// TIA Portal V16 export
// export: Created 2022-01-12T14:34:29.5419654Z, ExportSetting WithDefaults, DisplayName Totally Integrated Automation Portal, DisplayVersion V16 Update 4, DisplayName TIA Portal Version Control Interface, DisplayVersion V16 Update 2, DisplayName TIA Portal Openness, DisplayVersion V16 Update 4, DisplayName STEP 7 Professional, DisplayVersion V16 Update 4, DisplayName STEP 7 Safety, DisplayVersion V16, DisplayName WinCC Professional, DisplayVersion V16 Update 4
TYPE "typObiekt"
// stored: IsFailsafeCompliant false
   STRUCT
      typObiektu : Int := 1;
      nazwaObiektu : String[10] := 'F100AV01';
      procedura : Int;   // procedura 0 - to wyłaczenie/procedura 1 to załączenie
      inStartAuto : Bool;
      outStartUrządzenie : Bool;
      inLiftUp : Bool;
      outLiftUp : Bool;
      inLiftDown : Bool;
      outLiftDown : Bool;
      inZadaneWysterowanieAuto : Real;
      outWysterowanieUrządzenia : Real;
      inJestPotwWysterowania : Bool;
      diPotwWysterowania : Bool;
      inJestPotwNiewysterowania : Bool;
      diPotwNieWysterowania : Bool;
      inZezwolenieNaPracę : Bool;   // pkz+KSB+CKF+przełacznik wyłacznika siremontowego / z KSB
      Awaria : Bool;   // bit informujacy o awarii
      ResetAwaria : Bool;   // reset z programu
      kodBłedu : Word;   // kod statusu z urządzenia (falownik słowo statusu)
      czasDoAwariiSP : Int := 1000;
      czasDoAwariiPV : Int;
      czasPracyGodziny : Real;   // np. czas pracy pompy
      _ : Bool;
      hmiPokażStacyjkę : Bool;   // //stacyjka
      hmiStanUrządzenia : Int;   // rysunek na hmi
      hmiTrybAutoManual : Bool;   // zmiana trybu pracy urządzenia ze stacyjki
      hmiManualStart : Bool;   // /maualne załączenie pompy zaworu
      hmiManualStop : Bool;   // tylko żeby w stacujce pokazac przycisk/lampke
      hmiManualLiftUp : Bool;   // dla zaworów
      hmiManualLiftDown : Bool;   // dla zaworów
      hmiManualneWysterowanie : Real;   // /manualna wartosc analogowa ręka pompy /pida
      hmiSymulujSygnałyWejsciowe : Bool;   // załącz maskowanie/symulacje wejsc
      hmiSymulacjaPotwWysterowania : Bool;
      hmiSymulacjaPotwNieWysterowania : Bool;
      hmiSymulowanaWartośćAnalogowa : Real;   // symulowana wartość pomiarowa dla mierników
      hmiPotwNieWysterowania : Bool;
      hmiPotwWysterowania : Bool;   // wynikowy bit potwierdzenia wysterowania
      hmiZasilanieOK : Bool;   // potwierdzenie że termik załaczoony/ zasilanie falownika ok
      hmiResetAwaria : Bool;   // reset ze stacyjki
      hmiPrądFalownika : Real;   // prad falownika
      ___ : Bool;   // ////////////////////analogi///////////////////////
      inPomiarRaw : Int;   // wejście ai sterownika (0-27648) / pomiar
      minSkali : Real := -50.0;   // wartość dla 4mA - raw=0
      maxskali : Real := 150.0;   // wartość dla 20mA - raw 27648
      tFiltr : Real := 0.9;   // 0.8 -0.99 /d /rampa dla pompy 0 -99sekund
      pomiarTymczas : Real;
      wyjTymczas : Real;
      WartośćPomiaru : Real;   // pomiar analogowy
      ____ { ExternalWritable := 'False'} : Bool;   // ///////////////przepływomierz//////////////////////
      hmiMetry3NaImpuls : Real := 0.001;   // wartość nastawy dla wejścia impulsowego(jeżeli stosujemy)
      diImpulsy : Bool;   // wejście impulsowe z przepływomierza lub z programu
      R_Trig : Bool;   // impulsator z programu podczas załaczenia symulacji
      startLicznik1 : Bool;
      zerujLicznik1 : Bool;
      startLicznik2 : Bool;
      zerujLicznik2 : Bool;
      startLicznik3 : Bool;
      zerujLicznik3 : Bool;
      licznik1 : Real;
      licznik2 : Real;
      licznik3 : Real;
      licznikTotalImpulsy : Int;
      Lreal_1 : LReal;
      Lreal_2 : LReal;
      _____ : Bool;
      pid_SP : Real;   // //PID setpoint
      pid_PV : Real;   // proces value
      pid_P : Real := 1.0;
      pid_I : Real := 10.0;
      pid_D : Real;
      pid_Rampa : Real := 1.0;   // 0.0-1.0
      pid_Out : Real;
      ______ : Bool;
      SetReset { S7_SetPoint := 'True'} : "typSetReset";
      Flipaj : "typFlipaj";
      I1 { S7_SetPoint := 'True'} : Int;
      l2 : LReal;
      l4 : Word;
   END_STRUCT;
END_TYPE
